TYPE ST_MqttConfig :
STRUCT
	
	xEnable						: BOOL := FALSE;
	sHostName 					: STRING := 'localhost';
    nHostPort 					: UINT := 1883;
	
END_STRUCT
END_TYPE

(* stored: Version 1.1.0.1, ProductVersion 3.1.4024.12
   DUT ST_MqttConfig: Id {ac8a7c30-8bb4-4b32-ad2b-27c2fc7f9d2a} *)
